# EPICS substitutions: OLD/mc11/tpmacApp/Db/autohome.substitutions
file "$(EPICS_BASE)/db/autohome.db"
{

pattern
{SYS,              DEV,                 PLC,  PORT  }
{"XF:23ID2-BI",  "{Diag:3-Ax:Y}",      8     P0    }
}
